// TIA Portal V19 export
DATA_BLOCK "dbSysInfo"   // DB2
AUTHOR : CH
FAMILY : Aktina
NAME : Lib_System
// stored: AutoNumber false, InstanceOfName libCpu_SystemInfo, InstanceOfType FB
"libCpu_SystemInfo"
   // VAR_INPUT
   //    init { ExternalAccessible := 'False'; ExternalVisible := 'False'; ExternalWritable := 'False'} : Bool := FALSE;
   //    clockByte { ExternalWritable := 'False'} : Byte := 16#43;
   // END_VAR
   // VAR_OUTPUT
   //    timeByte { ExternalWritable := 'False'} : Byte := 16#01;
   //    localTime : DTL := DTL#2025-09-17-14:58:29.859354800;
   // END_VAR
   // VAR RETAIN
   //    statLocalTime { ExternalWritable := 'False'} : DTL := DTL#2025-09-17-14:58:29.769137900;
   //    statClockByteOld { ExternalWritable := 'False'} : Byte := 16#41;
   // END_VAR
   // VAR
   //    statTimeByte { ExternalWritable := 'False'} : Byte := 16#01;
   // END_VAR
BEGIN
END_DATA_BLOCK
